INTERFACE I_GenerateEvents

METHOD PUBLIC Off
VAR_INPUT
	EventName : T_MaxString;
	EventHandler : I_EventHandler;
END_VAR
END_METHOD

METHOD PUBLIC On
VAR_INPUT
	EventName : T_MaxString;
	EventHandler : I_EventHandler;
END_VAR
END_METHOD

END_INTERFACE

(* stored: Version 1.1.0.1, ProductVersion 3.1.4024.12
   Itf I_GenerateEvents: Id {adc70d30-6cf5-4528-9984-d9e34ac064b5}
   Method Off: Id {d8c1ff4d-8059-4022-9c70-cbb29824b7fc}
   Method On: Id {f68e4807-5613-450c-a5bc-1d788ab31d43} *)
